# EPICS autosave request: softglue/iocBoot/iocSoftGlue/auto_settings.req
file softGlue_SignalShow_settings.req  P=$(P) H=softGlue:
file softGlue_FPGAContent_settings.req P=$(P) H=softGlue:
file softGlue_FPGAInt_settings.req     P=$(P) H=softGlue:
file softGlue_convenience_settings.req     P=$(P) H=softGlue:

file softGlue_FPGAContent_octupole_settings.req   P=$(P) H=softGlue:
